PROGRAM POU_AxesError
VAR
	bAxis1ErrorI AT%I* :BOOL;
	bAxis2ErrorI AT%I* :BOOL;
	bAxis3ErrorI AT%I* :BOOL;
	bAxis4ErrorI AT%I* :BOOL;
	bAxis5ErrorI AT%I* :BOOL;
	bAxis6ErrorI AT%I* :BOOL;
END_VAR

IF bAxis1ErrorI OR bAxis2ErrorI OR bAxis3ErrorI OR bAxis4ErrorI OR bAxis5ErrorI OR bAxis6ErrorI
	THEN
	bMotorError:=FALSE;
	ELSE
		bMotorError:=TRUE;
END_IF

END_PROGRAM

(* stored: Version 1.1.0.1, ProductVersion 3.1.4022.18
   POU POU_AxesError: Id {14000388-cb1e-4082-ad11-428f6aceafb2}, SpecialFunc None *)
